FUNCTION_BLOCK Heating IMPLEMENTS I_Execute
VAR_INPUT
	bPumpOverload	: BOOL;
	bBoilerOverload	: BOOL;

	rBoilerTemp		: REAL;
	rBoilerPressure	: REAL;	
END_VAR
VAR_OUTPUT
	bPump			: BOOL;
	bBurner			: BOOL;
END_VAR
VAR
	_this			: Entity;
	_ctx			: Heating_Ctx;
	_tag			: Tag('Heating');
	_exe			: Execute(THIS^);
	
	_onEnable		: Signal;
	_compOnEnable	: Comp(_onEnable, _this);
	_proxOnEnable	: SignalProxy(_onEnable, _ctx.priv.iOnEnable);
	
	_onDisable		: Signal;
	_compOnDisable	: Comp(_onDisable, _this);
	_proxOnDisable	: SignalProxy(_onDisable, _ctx.priv.iOnDisable);
	
	_onPause		: Signal;
	_compOnPause	: Comp(_onPause, _this);
	_proxOnPause	: SignalProxy(_onPause, _ctx.priv.iOnPause);
	
	_onResume		: Signal;
	_compOnResume	: Comp(_onResume, _this);
	_proxOnResume	: SignalProxy(_onResume, _ctx.priv.iOnResume);
	
	_smgr			: StateManager<6>(_this);
	_proxSmgr		: StateManagerProxy(_smgr, _ctx.state.iMgr);
	
	_disabled		: Heating_State_Disabled(_this, _ctx);
	_proxDisabled	: StateProxy(_disabled, _ctx.state.iDisable);
	
	_safety			: Heating_State_Safety(_this, _ctx);
	_proxSafety		: StateProxy(_safety, _ctx.state.iSafety);
	
	_fault			: Heating_State_Fault(_this, _ctx);
	_proxFault		: StateProxy(_fault, _ctx.state.iFault);
	
	_enabled		: Heating_State_Enabled(_this, _ctx);
	_proxEnabled	: StateProxy(_enabled, _ctx.state.iEnable);
	
	_pumping		: Heating_State_Pumping(_this, _ctx);
	_proxPumping	: StateProxy(_pumping, _ctx.state.iPump);
	
	_heatup			: Heating_State_Heatup(_this, _ctx);
	_proxHeatup		: StateProxy(_heatup, _ctx.state.iHeatup);

	_passiveHeatingCount		: Heating_PassiveCountRec(_ctx);
	_passiveHeatingCountRec		: Receiver(_passiveHeatingCount);
	_compPassiveHeatingCountRec	: Comp(_passiveHeatingCountRec, _this);
	
	_request					: Heating_RequestRec(_ctx);
	_requestRec					: Receiver(_request);
	_compRequestRec				: Comp(_requestRec, _this);
	
	_queue						: ArgQueue<CST.MAX_PASSIVE_ROOM>;
	_queueProxy					: ArgQueueProxy(_queue, _ctx.priv.iQueue);
	
END_VAR

METHOD Execute
END_METHOD

END_FUNCTION_BLOCK

(* stored: Version 1.1.0.1
   POU Heating: Id {62f0b3a1-a792-4ec1-b14a-c56d60b72dc9}, SpecialFunc None
   Method Execute: Id {2db28cf4-24c2-48ef-813b-53c66671dd1a} *)
